FUNCTION_BLOCK MotorPOS (* Service Interface Function Block Type *)
  (* Standard: 61499-2 *)
  (* Version 0.0, 2012-06-03, 4DIAC-IDE, 4DIAC-Consortium *)
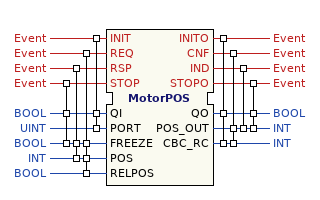
  EVENT_INPUT
    INIT WITH PORT, QI; (* Service Initialization *)
    REQ WITH POS, FREEZE, RELPOS; (* move to position request *)
    RSP WITH FREEZE, POS; (* Returns whether the motor has finished a move with specified position. *)
    STOP WITH QI, FREEZE;
  END_EVENT
  EVENT_OUTPUT
    INITO WITH QO, CBC_RC; (* Initialization Confirm *)
    CNF WITH POS_OUT, CBC_RC;
    IND WITH POS_OUT; (* specified position.reached *)
    STOPO WITH QO, POS_OUT;
  END_EVENT
  VAR_INPUT
    QI : BOOL; (* input qualifer *)
    PORT : UINT; (* Port the Motor is connected *)
    FREEZE : BOOL; (* when turn off then true freeze; false coast *)
    POS : INT; (* -1000 to 1000 ticks per second *)
    RELPOS : BOOL; (* Relative position = true; Absolute position = false *)
  END_VAR
  VAR_OUTPUT
    QO : BOOL; (* Event Output Qualifier; false if Port problem *)
    POS_OUT : INT;
    CBC_RC : INT;
  END_VAR
  SERVICE APPLICATION/RESOURCE (* Service Interface Function Block Type *)
    SEQUENCE normal_establishment
      APPLICATION.INIT+(PARAMS) -> APPLICATION.INITO+(PARAMS);
    END_SEQUENCE
    SEQUENCE unsuccessful_establishment
      APPLICATION.INIT+(PARAMS) -> APPLICATION.INITO-(STATUS);
    END_SEQUENCE
    SEQUENCE request_confirm
      APPLICATION.REQ+(SD) -> APPLICATION.CNF+(RD);
    END_SEQUENCE
    SEQUENCE request_inhibited
      APPLICATION.REQ-(SD) -> APPLICATION.CNF-(STATUS);
    END_SEQUENCE
    SEQUENCE request_error
      APPLICATION.REQ+(SD) -> APPLICATION.CNF-(STATUS);
    END_SEQUENCE
    SEQUENCE indication_response
      RESOURCE.indicate(RD) -> APPLICATION.IND+(RD);
      APPLICATION.RSP(QI,SD) -> RESOURCE.response(QI,SD);
    END_SEQUENCE
    SEQUENCE indication_inhibited
      RESOURCE.indicate(RD,QI=FALSE) -> RESOURCE.inhibited();
    END_SEQUENCE
    SEQUENCE error_indication
      RESOURCE.error(STATUS) -> APPLICATION.IND-(STATUS);
    END_SEQUENCE
    SEQUENCE application_initiated_termination
      APPLICATION.INIT-() -> APPLICATION.INITO-(STATUS);
    END_SEQUENCE
    SEQUENCE resource_initiated_termination
      -> APPLICATION.INITO-(STATUS);
    END_SEQUENCE
  END_SERVICE
END_FUNCTION_BLOCK
